(* PLC project PRG_AU_Acquisition_CFC.project, Dragage CODESYS CODESYS V3.5 SP19 Patch 1 *)
(* stored: creationDateTime 2026-08-01T00:00:00, modificationDateTime 2026-08-01T00:00:00 *)

(* Acquisition et qualification des entrees AU (CFC natif, cible AF02 §2). Lit les signaux simules (GVL_Simulation_AU) et les qualifie via FB_Input (brique standard, meme composant que PRG_00_Inputs) avant transmission au composite FB_Safety_EmergencyManagement. Aucune logique metier ici (regle TC-P02-002) : le feedback simulation est delegue a FB_Sim_AU_ChainFeedback, une page CFC ne fait qu'enchainer des blocs. Regle de cablage CFC (obligatoire, DOC/CODE_QUALITY_STANDARDS.md paragraphe CFC) : CHAQUE entree source (inVariable/sortie de bloc) passe par un connector dedie avant de rejoindre un bloc consommateur -- jamais de connexion directe source vers bloc. Chaque connector a une position UNIQUE et non nulle (x,y != 0,0 sauf le tout premier), pour eviter les fils de longueur nulle empiles qui rendent le cablage illisible/invisible dans l'editeur CODESYS (REX 2026-08). Docs : DOC/AF_Partie-01_Analyse_Fonctionnelle_v2.0.md DOC/AF_Partie-02_Architecture_Programme_v3.0.md §2 DOC/AF_Partie-06_Acquisition_Qualification_IO_v2.0.md *)
PROGRAM PRG_AU_Acquisition
  VAR_OUTPUT
    EmergencyChainClosed : BOOL;  (* Boucle AU fermee (qualifie FB_Input, 20 ms) *)
    PowerContactorEngaged : BOOL;  (* Contacteur puissance engage (qualifie FB_Input, 20 ms) *)
    PowerCutOffRequest : BOOL;  (* Demande coupure safety metier (agrege) *)
  END_VAR
  VAR
    instSimChainFeedback : FB_Sim_AU_ChainFeedback;  (* Simulation physique boucle AU (banc de test) *)
    instEmergencyChainClosed : FB_Input;  (* Qualification boucle AU (anti-rebond 20 ms) *)
    instPowerContactorEngaged : FB_Input;  (* Qualification retour contacteur (anti-rebond 20 ms) *)
  END_VAR

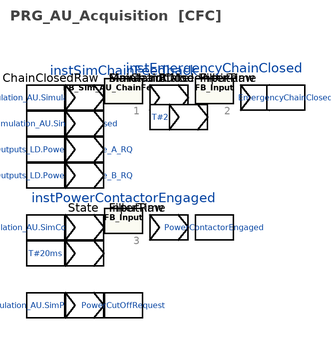
(* CFC diagram, written out as Structured Text *)
instSimChainFeedback(SimulationModeActive := GVL_Simulation_AU.SimulationModeActive, SimChainClosed := GVL_Simulation_AU.SimChainClosed, MaintainA := PRG_AU_Outputs_LD.PowerKeepAlive_A_RQ, MaintainB := PRG_AU_Outputs_LD.PowerKeepAlive_B_RQ);
instEmergencyChainClosed(InputRaw := instSimChainFeedback.ChainClosedRaw, FilterTime := T#20ms);
instPowerContactorEngaged(InputRaw := GVL_Simulation_AU.SimContactorEngaged, FilterTime := T#20ms);
EmergencyChainClosed := instEmergencyChainClosed.State;
PowerContactorEngaged := instPowerContactorEngaged.State;
PowerCutOffRequest := GVL_Simulation_AU.SimPowerCutOffReq;
END_PROGRAM
